// TIA Portal V18 export
TYPE "LGasp_typeStatoAttuatore"
// stored: IsFailsafeCompliant false
   STRUCT
      qatt : LReal;   // quota attuale
      tatt : LReal;   // torque attuale
      satt : LReal;   // velocita attuale
      fcpos : Bool;   // posizione positiva
      fcneg : Bool;   // posizione negativa
      flt : Bool;   // Attuatore in errore
      peh : Bool;   // Attuatore in PEH
      timepos : Time := T#0MS;   // Tempo posizionamento avanti
      timeneg : Time := T#0MS;   // Tempo posizionamento indietro
   END_STRUCT;
END_TYPE
